// Mitsubishi GX Works2 project: IELET2103_Datalab5   PLC: FX2N/FX2NC
// IELET2103_Datalab5

// global labels: Global1
VAR_GLOBAL
  BarnInn AT X000 : BOOL;
  VoksenInn AT X001 : BOOL;
  BarnUt AT X002 : BOOL;
  VoksenUt AT X003 : BOOL;
  Nullstill AT X010 : BOOL;
  AntBarnInne AT D0 : WORD;
  AntVoksneInne AT D2 : WORD;
  AntPersInne AT D4 : WORD;
  TotAntBarn AT D6 : WORD;
END_VAR
VAR_GLOBAL CONSTANT
  PrisBarn : WORD := 75;
  PrisVoksen : WORD := 100;
END_VAR
VAR_GLOBAL
  DagsInntektBarn AT D20 : DWORD;
  DagsInntektVoksen AT D22 : DWORD;
  DagsInntektTotal AT D24 : DWORD;
  TotAntVoksne AT D8 : WORD;
  InntektDagerBarn AT D100 : ARRAY [0..49] OF DINT;
  InntektDagerVoksen AT D200 : ARRAY [0..49] OF DINT;
END_VAR

// task Task_01 (event TRUE, interval 0, priority 31): POU_01

PROGRAM POU_01
(* structured ladder/FBD written out as ST: instructions are called as NAME(EN, inputs, outputs); _pN, _eN, _tN stand for wires *)
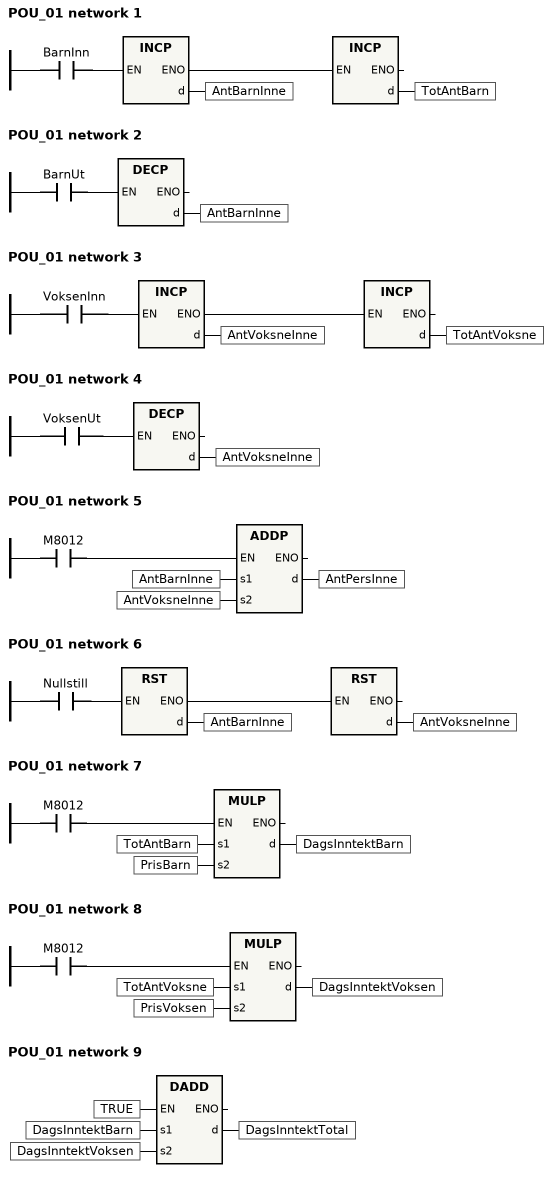
(* network 1 *)
_e1 := INCP(BarnInn, AntBarnInne);
INCP(_e1, TotAntBarn);
(* network 2 *)
DECP(BarnUt, AntBarnInne);
(* network 3 *)
_e1 := INCP(VoksenInn, AntVoksneInne);
INCP(_e1, TotAntVoksne);
(* network 4 *)
DECP(VoksenUt, AntVoksneInne);
(* network 5 *)
ADDP(M8012, AntBarnInne, AntVoksneInne, AntPersInne);
(* network 6 *)
_e1 := RST(Nullstill, AntBarnInne);
RST(_e1, AntVoksneInne);
(* network 7 *)
MULP(M8012, TotAntBarn, PrisBarn, DagsInntektBarn);
(* network 8 *)
MULP(M8012, TotAntVoksne, PrisVoksen, DagsInntektVoksen);
(* network 9 *)
DADD(TRUE, DagsInntektBarn, DagsInntektVoksen, DagsInntektTotal);
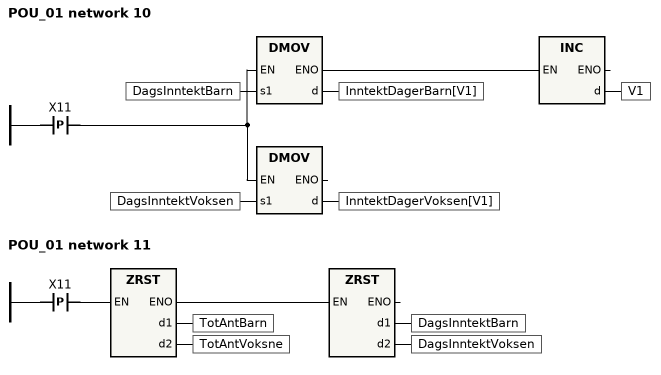
(* network 10 *)
_p1 := LDP(TRUE, X11);
_e2 := DMOV(_p1, DagsInntektBarn, InntektDagerBarn[V1]);
INC(_e2, V1);
DMOV(_p1, DagsInntektVoksen, InntektDagerVoksen[V1]);
(* network 11 *)
_e1 := ZRST(LDP(TRUE, X11), TotAntBarn, TotAntVoksne);
ZRST(_e1, DagsInntektBarn, DagsInntektVoksen);
END_PROGRAM

FUNCTION_BLOCK Dagslogg
;
END_FUNCTION_BLOCK
